PROGRAM XML
VAR
   savedvalues     : ST_SavedStructure;
   fbXmlSrvWrite   : FB_XmlSrvWrite;
   fbXmlSrvRead    : FB_XmlSrvRead; 
   sFileFolder     : T_MaxString := '\Hard Disk\'; (* CE: '\Hard Disk\' *) (* Win10: '\C:\ *)
   sFileName       : T_MaxString := 'HMI-Saved-Positions.xml';
   //sFilePath 	   : T_MaxString := 'C:\HMI-Saved-Positions.xml';  				//disable for CE
   sFilePath       : T_MaxString := '\Hard Disk\HMI-Saved-Positions.xml';		//enable for CE
   (*sFilePathWrite = sFileFolder + time + sFileName*)
   bExecute        : BOOL; 
   sXPath          : T_MaxString := '/dataentry/MAIN.savedvalues';
   ntGetTime       : NT_GetTime;
   stMyTimestruct  : TIMESTRUCT;
   iState          : INT := 0;
   bTwentySec      : BOOL:= FALSE;
   bButton         : BOOL:= FALSE;
   bTwentySecOver  : BOOL;
   triggerWrite    : R_TRIG;
   triggerButton   : R_TRIG;
   i			   : INT:=1;
   LoadComplete   : BOOL;
END_VAR

triggerButton(CLK:= bButton);


CASE iState OF
0: (* initialize *)
   fbXmlSrvRead(
   	 pSymAddr  := ADR(savedvalues),
     cbSymSize := SIZEOF(savedvalues), 
     sFilePath := sFilePath,
     sXPath    := sXPath,
     bExecute  := TRUE
   );
   iState:= 1; 
   ;
   
1: (* wait for read operation *)
   fbXmlSrvRead(bExecute:= FALSE);
   IF NOT fbXmlSrvRead.bBusy AND NOT fbXmlSrvRead.bError THEN
     iState:= 2; 
	 LoadComplete := TRUE;
   ELSIF fbXmlSrvRead.bError THEN
     iState:= 100;
	 LoadComplete:=FALSE;
   END_IF
 
2: (* Write *)
	savedvalues.counter:=savedvalues.counter + 1;
	IF savedvalues.counter = 326767 THEN
		savedvalues.counter := 0;
	END_IF

   fbXmlSrvWrite(nMode:=XMLSRV_ADDMISSING, pSymAddr:= ADR(savedvalues),
   cbSymSize:= SIZEOF(savedvalues));
   ntGetTime(START:= TRUE, TIMESTR=>stMyTimestruct); (* get Windows time *)
   IF NOT ntGetTime.BUSY AND NOT ntGetTime.ERR THEN
      iState:= 5;
   ELSIF ntGetTime.ERR THEN
      iState:= 100;
 END_IF
   
5: (* working state *)
   ntGetTime(START:= FALSE);
   IF NOT ntGetTime.BUSY AND NOT ntGetTime.ERR THEN
      ntGetTime(START:= TRUE, TIMESTR=>stMyTimestruct);
   ELSIF ntGetTime.ERR THEN
      iState:= 100;
   END_IF

	IF stMyTimestruct.wMinute = 0 OR stMyTimestruct.wMinute = 15 OR stMyTimeStruct.wMinute = 30 OR stMyTimeStruct.wMinute = 45 OR stMyTimeStruct.wMinute = 60 THEN
		bTwentySecOver:= TRUE;
		savedvalues.rStagePosition := GV_LIFT.STAGE_POSITION;
	ELSE
		bTwentySecOver:= FALSE;
	END_IF
	
   (* if 20s have passed => trigger writing-process *)
   triggerWrite(CLK:=bTwentySecOver);
   IF (triggerWrite.Q OR triggerButton.Q) AND NOT fbXmlSrvWrite.bBusy AND NOT fbXmlSrvWrite.bError THEN 
      (* write *)
      fbXmlSrvWrite(sFilePath:=sFilePath, sXPath:=sXPath, bExecute:= TRUE);

   ELSIF fbXmlSrvWrite.bError THEN
      iState:= 100;
   END_IF

   (* reset fbXmlSrvWrite *)
   IF fbXmlSrvWrite.bBusy AND NOT ntGetTime.ERR THEN
      fbXmlSrvWrite(bExecute:= FALSE);
   ELSIF ntGetTime.ERR THEN
      iState:= 100;
   END_IF
 
100: (* error state*) 
 ;

END_CASE

END_PROGRAM

(* stored: Version 1.1.0.1, ProductVersion 3.1.4022.12
   POU XML: Id {6eef0ea7-4544-4415-8d0d-0f64a62ae60c}, SpecialFunc None *)
